PROGRAM GarageDoor
VAR
	fbMotion : MoveGarageDoor;
	bActuationButton AT %I* : BOOL; //button that we control through visualization
	bErrorButton AT %I* : BOOL; //button for simulating error
	bDoorOpened : BOOL; //sensor for open door
	bDoorClosed : BOOL; //sensor for close door
	bDoorDriveOverload : BOOL; //sensor for the overload of the door
	bDoorPaused : BOOL; //sensor for pausing the door
	bMotionLight : BOOL; //light that indicates there is motion
	fPosition : LREAL; //shows the position of the door
	
	bTest1 : BOOL;
	bTest2 : BOOL;
	bTest3 : BOOL;
	
	bTest4 : BOOL;
	bTest5 : BOOL;
	
	bPauseVis : BOOL;
	bErrorVis : BOOL;

END_VAR

fbMotion.bActuationProgram := bActuationButton;
fbMotion.bError := bErrorButton;

bDoorOpened := fbMotion.bOpened;
bDoorClosed := fbMotion.bClosed;
bDoorDriveOverload := fbMotion.bDriveOverload;
bDoorPaused := fbMotion.bPaused;
bMotionLight := fbMotion.bLight;

fPosition := fbMotion.fActPos;

bTest1 := fbMotion.bVis1O;
bTest2 := fbMotion.bVis2O;
bTest3 := fbMotion.bVis3O;

bTest4 := fbMotion.bVis1C;
bTest5 := fbMotion.bVis2C;

bPauseVis := fbMotion.bPauseImg;
bErrorVis := fbMotion.bErrorImg;


fbMotion();

END_PROGRAM

(* stored: Version 1.1.0.1, ProductVersion 3.1.4024.12
   POU GarageDoor: Id {61d642d1-b05b-46ad-9be9-dc37a7c45005}, SpecialFunc None *)
